FUNCTION_BLOCK client (* Tamplate for a simple Basic Function Block Type *)
  (* Standard: 61499-2 *)
  (* Version 0.0, 2018-01-28, 4DIAC-IDE, 4DIAC-Consortium *)
  (* Version 1.0, 2016-05-26, AZ, fortiss GmbH *)
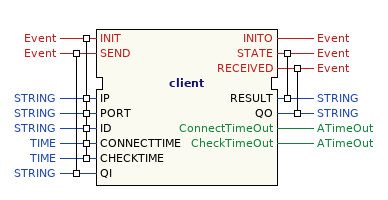
  EVENT_INPUT
    INIT WITH IP, PORT, ID, CONNECTTIME, CHECKTIME; (* Initialization Request *)
    SEND WITH QI; (* Normal Execution Request *)
  END_EVENT
  EVENT_OUTPUT
    INITO; (* Initialization Confirm *)
    STATE WITH RESULT;
    RECEIVED WITH QO; (* Execution Confirmation *)
  END_EVENT
  VAR_INPUT
    IP : STRING;
    PORT : STRING;
    ID : STRING;
    CONNECTTIME : TIME;
    CHECKTIME : TIME;
    QI : STRING; (* Input event qualifier *)
  END_VAR
  VAR_OUTPUT
    RESULT : STRING;
    QO : STRING; (* Output event qualifier *)
  END_VAR
  PLUGS
    ConnectTimeOut : ATimeOut;
    CheckTimeOut : ATimeOut;
  END_PLUGS
  VAR
    ISCONNECT : BOOL := FALSE; (* Internal Variable *)
    ISNOTICE : BOOL := FALSE; (* Internal Variable *)
  END_VAR
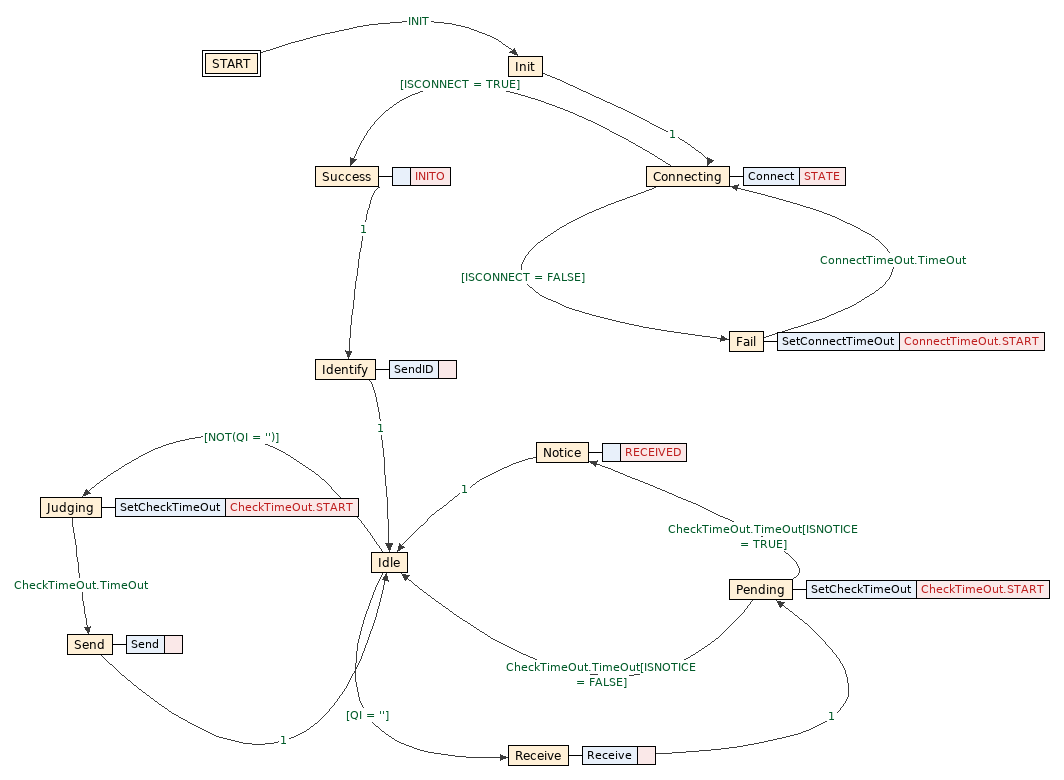
  EC_STATES
    START; (* Initial State *)
    Init;
    Idle;
    Send : Send;
    Receive : Receive;
    Success : -> INITO;
    Connecting : Connect -> STATE;
    Pending : SetCheckTimeOut -> CheckTimeOut.START;
    Notice : -> RECEIVED;
    Fail : SetConnectTimeOut -> ConnectTimeOut.START;
    Identify : SendID;
    Judging : SetCheckTimeOut -> CheckTimeOut.START;
  END_STATES
  EC_TRANSITIONS
    START TO Init := INIT;
    Init TO Connecting := 1;
    Connecting TO Success := [ISCONNECT = TRUE];
    Receive TO Pending := 1;
    Pending TO Notice := CheckTimeOut.TimeOut[ISNOTICE = TRUE];
    Notice TO Idle := 1;
    Pending TO Idle := CheckTimeOut.TimeOut[ISNOTICE = FALSE];
    Connecting TO Fail := [ISCONNECT = FALSE];
    Fail TO Connecting := ConnectTimeOut.TimeOut;
    Success TO Identify := 1;
    Send TO Idle := 1;
    Idle TO Receive := [QI = ''];
    Identify TO Idle := 1;
    Idle TO Judging := [NOT(QI = '')];
    Judging TO Send := CheckTimeOut.TimeOut;
  END_TRANSITIONS
  ALGORITHM Connect IN ST: (* new algorithm *)

  END_ALGORITHM
  ALGORITHM Send IN ST: (* new algorithm *)

  END_ALGORITHM
  ALGORITHM Receive IN ST: (* new algorithm *)

  END_ALGORITHM
  ALGORITHM SendID IN ST: (* new algorithm *)

  END_ALGORITHM
  ALGORITHM SetConnectTimeOut IN ST: (* new algorithm *)
ConnectTimeOut.DT := CONNECTTIME;
  END_ALGORITHM
  ALGORITHM SetCheckTimeOut IN ST: (* new algorithm *)
CheckTimeOut.DT := CHECKTIME;
  END_ALGORITHM
END_FUNCTION_BLOCK
